Fanuc TP program (LS listing): BG_STATUS.LS

/PROG  BG_STATUS
/ATTR
OWNER		= MNEDITOR;
COMMENT		= "";
PROG_SIZE	= 184;
CREATE		= DATE 21-08-29  TIME 13:29:06;
MODIFIED	= DATE 21-08-29  TIME 13:29:42;
FILE_NAME	= ;
VERSION		= 0;
LINE_COUNT	= 0;
MEMORY_SIZE	= 428;
PROTECT		= READ_WRITE;
TCD:  STACK_SIZE	= 0,
      TASK_PRIORITY	= 50,
      TIME_SLICE	= 0,
      BUSY_LAMP_OFF	= 0,
      ABORT_REQUEST	= 0,
      PAUSE_REQUEST	= 0;
DEFAULT_GROUP	= *,*,*,*,*;
CONTROL_CODE	= 00000000 00000000;
LOCAL_REGISTERS	= 20,0,0;
/APPL

AUTO_SINGULARITY_HEADER;
  ENABLE_SINGULARITY_AVOIDANCE   : FALSE;
/MN
/POS
/END
